{attribute addProperty BoxType "EL3314-0010-0016"}
{attribute addProperty Id "TC_Inputs_ChannelAT %I*ARRAY[0..3] OF TC_Inputs_Channel_842FAF6F50062.50WcStateAT %I*WcState_F855686C1620InfoDataAT %I*InfoData_BC63D37F80100"}
{attribute addProperty CRC "83103709"}
{attribute addProperty SizeInBites "596"}
{attribute addProperty SizeInBytes "74.5"}
TYPE EL3314_2530FC31 :
STRUCT
	{attribute addProperty Name "TC_Inputs_Channel"}
	TC_Inputs_Channel : ARRAY[0..3] OF TC_Inputs_Channel_842FAF6F;
	{attribute addProperty Name "WcState"}
	WcState : WcState_F855686C;
	{attribute addProperty Name "InfoData"}
	InfoData : InfoData_BC63D37F;
END_STRUCT
END_TYPE

(* stored: Version 1.2.0.0, ProductVersion 3.1.4024.9
   DUT EL3314_2530FC31: Id {523daf37-ce00-4df0-be28-1a92789ba5e1} *)
